% RSLogix 500 project TANK_CONTROL_BAK002.RSS, saved by version 8.30.00.16 %
PROJECT "UNTITLED"    % processor: Bul.1763 MicroLogix 1100 Series B %

PROGRAM FILES
  LAD 2 "MAIN"  4 rungs
  LAD 3 "DIGITAL IO"  7 rungs
  LAD 4 "CONTROLS"  6 rungs
  LAD 5 "ANALOG IO"  2 rungs

DATA FILES
  O0 OUTPUT  7 elements
  I1 INPUT  13 elements
  S2 STATUS  66 elements
  B3 BINARY  1 elements
  T4 TIMER  2 elements
  C5 COUNTER  1 elements
  R6 CONTROL  1 elements
  N7 INTEGER  1 elements
  F8 FLOAT  2 elements

LADDER 2 "MAIN"
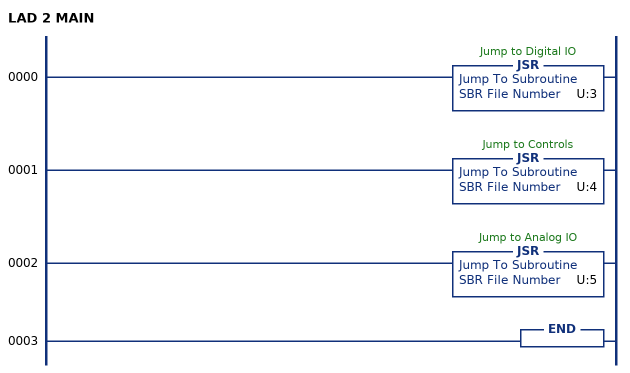
% Rung: 0 %
SOR JSR U:3 EOR
%   U:3  "Jump to Digital IO" %
% Rung: 1 %
SOR JSR U:4 EOR
%   U:4  "Jump to Controls" %
% Rung: 2 %
SOR JSR U:5 EOR
%   U:5  "Jump to Analog IO" %
% Rung: 3 %
SOR END EOR

LADDER 3 "DIGITAL IO"
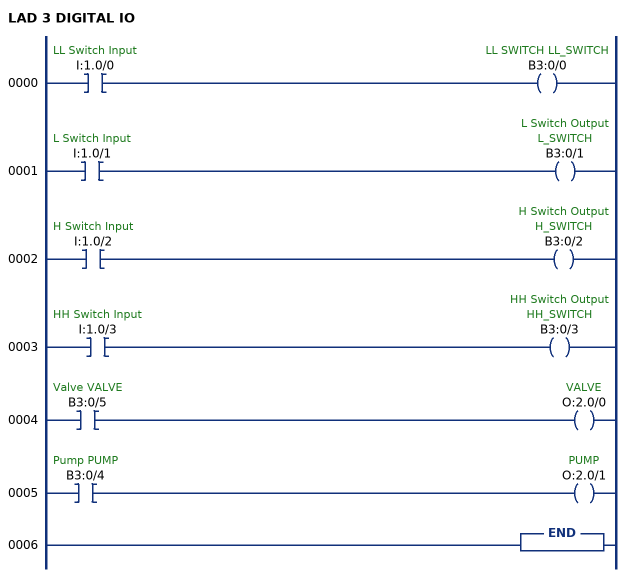
% Rung: 0 %
SOR XIC I:1.0/0 OTE B3:0/0 EOR
%   I:1.0/0  "LL Switch Input" %
%   B3:0/0  LL_SWITCH  "LL SWITCH" %
% Rung: 1 %
SOR XIC I:1.0/1 OTE B3:0/1 EOR
%   I:1.0/1  "L Switch Input" %
%   B3:0/1  L_SWITCH  "L Switch Output" %
% Rung: 2 %
SOR XIC I:1.0/2 OTE B3:0/2 EOR
%   I:1.0/2  "H Switch Input" %
%   B3:0/2  H_SWITCH  "H Switch Output" %
% Rung: 3 %
SOR XIC I:1.0/3 OTE B3:0/3 EOR
%   I:1.0/3  "HH Switch Input" %
%   B3:0/3  HH_SWITCH  "HH Switch Output" %
% Rung: 4 %
SOR XIC B3:0/5 OTE O:2.0/0 EOR
%   B3:0/5  VALVE  "Valve" %
%   O:2.0/0  "VALVE" %
% Rung: 5 %
SOR XIC B3:0/4 OTE O:2.0/1 EOR
%   B3:0/4  PUMP  "Pump" %
%   O:2.0/1  "PUMP" %
% Rung: 6 %
SOR END EOR

LADDER 4 "CONTROLS"
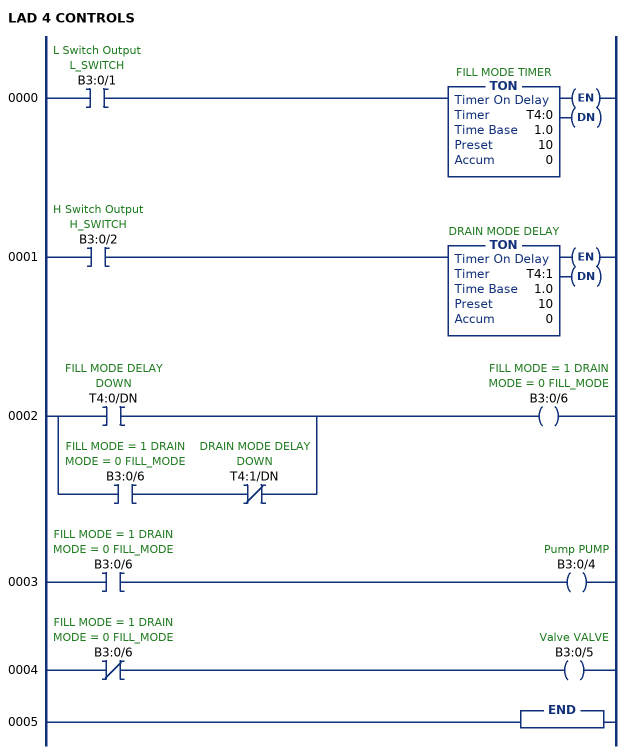
% Rung: 0 %
SOR XIC B3:0/1 TON T4:0 1.0 10 0 EOR
%   B3:0/1  L_SWITCH  "L Switch Output" %
%   T4:0  "FILL MODE TIMER" %
% Rung: 1 %
SOR XIC B3:0/2 TON T4:1 1.0 10 0 EOR
%   B3:0/2  H_SWITCH  "H Switch Output" %
%   T4:1  "DRAIN MODE DELAY" %
% Rung: 2 %
SOR BST XIC T4:0/DN NXB XIC B3:0/6 XIO T4:1/DN BND OTE B3:0/6 EOR
%   T4:0/DN  "FILL MODE DELAY DOWN" %
%   B3:0/6  FILL_MODE  "FILL MODE = 1 DRAIN MODE = 0" %
%   T4:1/DN  "DRAIN MODE DELAY DOWN" %
% Rung: 3 %
SOR XIC B3:0/6 OTE B3:0/4 EOR
%   B3:0/6  FILL_MODE  "FILL MODE = 1 DRAIN MODE = 0" %
%   B3:0/4  PUMP  "Pump" %
% Rung: 4 %
SOR XIO B3:0/6 OTE B3:0/5 EOR
%   B3:0/6  FILL_MODE  "FILL MODE = 1 DRAIN MODE = 0" %
%   B3:0/5  VALVE  "Valve" %
% Rung: 5 %
SOR END EOR

LADDER 5 "ANALOG IO"
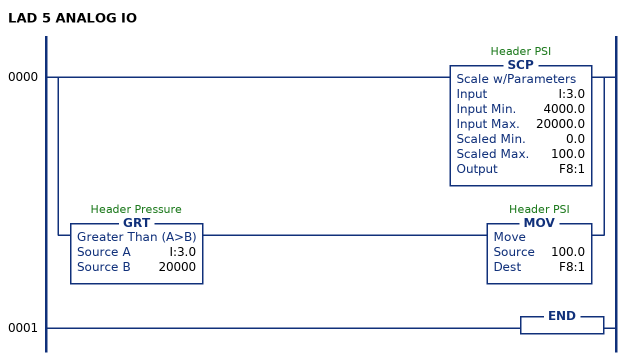
% Rung: 0 %
SOR BST SCP I:3.0 4000.0 20000.0 0.0 100.0 F8:1 NXB GRT I:3.0 20000 MOV 100.0 F8:1 BND EOR
%   I:3.0  "Header Pressure" %
%   F8:1  "Header PSI" %
% Rung: 1 %
SOR END EOR

REVISION NOTES
  0: digital io
  1: finished controls
  2: controls

DATA TABLE (non-zero values as saved)
DATA T4
% .PRE .ACC %
% T4:0 % 10 0
% T4:1 % 10 0
